// TIA Portal V17 export
// export: Created 2022-01-26T16:43:15.0076192Z, ExportSetting WithDefaults, DisplayName Totally Integrated Automation Portal, DisplayVersion V17, DisplayName TIA Portal Openness, DisplayVersion V17, DisplayName TIA Portal Version Control Interface, DisplayVersion V17, DisplayName STEP 7 Professional, DisplayVersion V17, DisplayName STEP 7 Safety, DisplayVersion V17, DisplayName WinCC Professional, DisplayVersion V17
DATA_BLOCK "NodeRed"   // DB4
{ S7_Optimized_Access := 'FALSE' }
VERSION : 0.1
// stored: AutoNumber true, DBAccessibleFromOPCUA true, DBAccessibleFromWebserver true, IsOnlyStoredInLoadMemory false, IsWriteProtectedInAS false
   VAR
      motorHusilloON : Bool;
      pidON : Bool;
      paro : Bool;
      triggerCMD : Bool;
      gramosSiwarex : Int;
      setpoint : Int;
      variadorHzFrecuenciaAuto : Int;
      variadorHzFrecuenciaManual : Int;
      variadorHzFrecuenciaSalida : Int;
      errorMin : Int := 10;
      cmdSiwarex : Int;
   END_VAR
BEGIN
END_DATA_BLOCK
